(* IEC 61131-3 sources: xPLCCore/codesys_code/Application/COMM_FBs/FB_RingBufferIndex, 18 files *)

(* ---- FB_RingBufferIndex.st ---- *)
(*
    Function Block: FB_RingBufferIndex
    Description:    Manages the indices of a ring (circular) buffer.
                    This FB does not store any data itself, but rather provides the correct
                    indices for an external data buffer array.

    Behavior:
    - 'Head' (H): The index where the NEXT new element should be written.
    - 'Tail' (T): The index of the OLDEST element that can be read.

    Visualization:
    | . . . . . T . . . . . H . . . . . |
                ^           ^
                |           |
             Oldest Data   Next Write Slot

    SPSC lock-free safety (added 2026-04-27):
    - Producer task is the only writer of _head (via PushHead).
    - Consumer task is the only writer of _tail (via ConsumeTail).
    - size() / space() are *derived* from _head and _tail; no _count
      RMW that both sides would race on.
    - _head / _tail count modulo (2 * _capacity) to disambiguate empty
      from full without sacrificing a slot. Slot index is recovered as
      (_head MOD _capacity) / (_tail MOD _capacity).
    - UINT reads/writes are single-instruction on the underlying CPU
      (16-bit aligned), so a stale cross-task read produces a
      conservative miss (false-full at the producer, false-empty at the
      consumer) that self-corrects on the next scan.
    - clear() writes both _head and _tail and is therefore NOT
      preemption-safe; only call it from a single-task context (init or
      offline-only), never from inside a producer/consumer loop.

    NOT MPSC-safe: if two tasks both push (or both consume) on the same
    instance, GetHead() can return the same slot to both producers and
    PushHead() can race on _head. In this project reMP_info_ridx is
    pushed only by EC_Task (AxisGroupSM family) and consumed only by
    Comm task (TCP_MSGPAK_Server) -- a clean SPSC arrangement. Earlier
    revisions had EC_Task perform ConsumeTail() on overflow ("drop-
    oldest") which created a second consumer racing the Comm task; that
    has been replaced everywhere with a "drop-newest" pattern (skip the
    write if space()=0, or pack into GVL.reMP_info_scratch and decline
    to PushHead). See doc/3-subsystems/ringbuf-bugs.md item #12.

    Author:         Gemini (initial), refactored to SPSC lock-free 2026-04-27
    Version:        2.0
*)
FUNCTION_BLOCK FB_RingBufferIndex
VAR_INPUT
END_VAR
VAR_OUTPUT
END_VAR
VAR
    // Internal state variables. _head is producer-owned; _tail is
    // consumer-owned. Each is updated by a single task only.
    _head           : UINT := 0;   // Next write position, mod _cap2.
    _tail           : UINT := 0;   // Next read position,  mod _cap2.
    _capacity       : UINT := 0;   // User-visible capacity (set by init()).
    _cap2           : UINT := 0;   // _capacity * 2, precomputed for size math.
END_VAR
(* =========== IMPLEMENTATION =========== *)

(* ---- Capacity.st ---- *)
METHOD Capacity : UINT
VAR_INPUT
END_VAR
(* =========== IMPLEMENTATION =========== *)
Capacity := _capacity;

(* ---- capacity.st ---- *)
METHOD capacity : UINT
VAR_INPUT
END_VAR
(* =========== IMPLEMENTATION =========== *)
capacity := _capacity;

(* ---- Clear.st ---- *)
METHOD Clear : BOOL
VAR_INPUT
END_VAR
(* =========== IMPLEMENTATION =========== *)
// Writes both _head and _tail. Not safe under task preemption -- only
// call from a single-task context (init or offline). The legacy
// in-loop clear() in AxisGroupSM was removed when the not-Ready drain
// path switched to per-packet NAK.
_head := 0;
_tail := 0;

(* ---- clear.st ---- *)
METHOD clear : BOOL
VAR_INPUT
END_VAR
(* =========== IMPLEMENTATION =========== *)
_head := 0;
_tail := 0;
_count := 0;

(* ---- ConsumeTail.st ---- *)
METHOD ConsumeTail : BOOL
VAR_INPUT
END_VAR
(* =========== IMPLEMENTATION =========== *)
    IF Size() = 0 THEN
        ConsumeTail := FALSE; // Buffer empty
        RETURN;
    END_IF;

    // Consumer-only write; producer observes the new tail and learns a
    // slot freed up.
    _tail := (_tail + 1) MOD _cap2;

    ConsumeTail := TRUE;

(* ---- consumeTail.st ---- *)
METHOD consumeTail : BOOL
VAR_INPUT
END_VAR
(* =========== IMPLEMENTATION =========== *)
    IF size() = 0 THEN
        consumeTail := FALSE; // Buffer empty
        RETURN;
    END_IF;

    // Consumer-only write; producer observes the new tail and learns a
    // slot freed up.
    _tail := (_tail + 1) MOD _cap2;

    consumeTail := TRUE;

(* ---- FB_init.st ---- *)
METHOD FB_init : BOOL
VAR_INPUT
    bInitRetains : BOOL; // This input is required by the FB_init standard but not used here.
    bInCopyCode  : BOOL; // This input is required by the FB_init standard but not used here.
    ring_buffer_size : UINT; // The total capacity of the buffer
END_VAR
(* =========== IMPLEMENTATION =========== *)

FB_init:=init(ring_buffer_size);

(* ---- GetHead.st ---- *)
METHOD GetHead : DINT
(* =========== IMPLEMENTATION =========== *)

    // Full check via derived size; safer than read-modify-write _count.
    IF Size() >= _capacity THEN
        GetHead := -1; // Buffer full
        RETURN;
    END_IF;

    // External slot index lives in [0.._capacity-1]; internal _head
    // lives in [0.._cap2-1] for empty/full disambiguation.
    GetHead := UINT_TO_DINT(_head MOD _capacity);

(* ---- getHead.st ---- *)
METHOD getHead : DINT
(* =========== IMPLEMENTATION =========== *)

    // Full check via derived size; safer than read-modify-write _count.
    IF size() >= _capacity THEN
        getHead := -1; // Buffer full
        RETURN;
    END_IF;

    // External slot index lives in [0.._capacity-1]; internal _head
    // lives in [0.._cap2-1] for empty/full disambiguation.
    getHead := UINT_TO_DINT(_head MOD _capacity);

(* ---- GetTail.st ---- *)
METHOD GetTail : DINT
VAR_INPUT
END_VAR
(* =========== IMPLEMENTATION =========== *)
    IF Size() = 0 THEN
        GetTail := -1; // Buffer empty
        RETURN;
    END_IF;

    GetTail := UINT_TO_DINT(_tail MOD _capacity);

(* ---- getTail.st ---- *)
METHOD getTail : DINT
VAR_INPUT
END_VAR
(* =========== IMPLEMENTATION =========== *)
    // Check for initialization and if there are items to consume
    IF (_count = 0) THEN
        getTail := -1; // Return -1 to indicate buffer is empty or not ready
        RETURN;
    END_IF;

    getTail := UINT_TO_DINT(_tail);

(* ---- init.st ---- *)
METHOD init : BOOL
VAR_INPUT
    ring_buffer_size : UINT; // The total capacity of the buffer
END_VAR
(* =========== IMPLEMENTATION =========== *)

_head := 0;
_tail := 0;
_capacity := ring_buffer_size;
// Pointer arithmetic happens modulo _cap2 so empty (head==tail) is
// distinct from full (size==_capacity). UINT max=65535; safe for any
// ring_buffer_size up to 32767.
_cap2 := ring_buffer_size * 2;

IF ring_buffer_size = 0 THEN
    // Buffer capacity cannot be zero.
    init := FALSE;
    RETURN;
END_IF;

init := TRUE;

(* ---- PushHead.st ---- *)
METHOD PushHead : BOOL
VAR_INPUT
END_VAR
(* =========== IMPLEMENTATION =========== *)

    IF Size() >= _capacity THEN
        PushHead := FALSE; // Buffer full
        RETURN;
    END_IF;

    // Producer-only write; pairs with the producer's prior data write
    // into slot[GetHead()]. Consumer observes the new head and only
    // then dereferences the slot.
    _head := (_head + 1) MOD _cap2;

    PushHead := TRUE;

(* ---- pushHead.st ---- *)
METHOD pushHead : BOOL
VAR_INPUT
END_VAR
(* =========== IMPLEMENTATION =========== *)

    IF size() >= _capacity THEN
        pushHead := FALSE; // Buffer full
        RETURN;
    END_IF;

    // Producer-only write; pairs with the producer's prior data write
    // into slot[getHead()]. Consumer observes the new head and only
    // then dereferences the slot.
    _head := (_head + 1) MOD _cap2;

    pushHead := TRUE;

(* ---- Size.st ---- *)
METHOD Size : UINT
VAR
    h : UINT;
    t : UINT;
END_VAR
(* =========== IMPLEMENTATION =========== *)
// Snapshot _head and _tail once. Each is single-task-owned and a UINT
// read is atomic on the CPU, so a stale cross-task read is at worst
// slightly conservative (a producer underestimates space for one scan,
// a consumer underestimates queued items for one scan). Both
// self-correct on the next call.
h := _head;
t := _tail;
IF h >= t THEN
    Size := h - t;
ELSE
    Size := h + _cap2 - t;
END_IF;

(* ---- size.st ---- *)
METHOD size : UINT
VAR
    h : UINT;
    t : UINT;
END_VAR
(* =========== IMPLEMENTATION =========== *)
// Snapshot _head and _tail once. Each is single-task-owned and a UINT
// read is atomic on the CPU, so a stale cross-task read is at worst
// slightly conservative (a producer underestimates space for one scan,
// a consumer underestimates queued items for one scan). Both
// self-correct on the next call.
h := _head;
t := _tail;
IF h >= t THEN
    size := h - t;
ELSE
    size := h + _cap2 - t;
END_IF;

(* ---- space.st ---- *)
METHOD space : UINT
VAR_INPUT
END_VAR
(* =========== IMPLEMENTATION =========== *)
space := _capacity - _count;
